SUBAPPLICATION Counter (* Subapplication Type *)
  (* Standard: 61499-2 *)
  (* Version 1.0, 2023-02-17, Franz *)
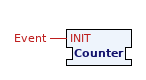
  EVENT_INPUT
    INIT;
  END_EVENT
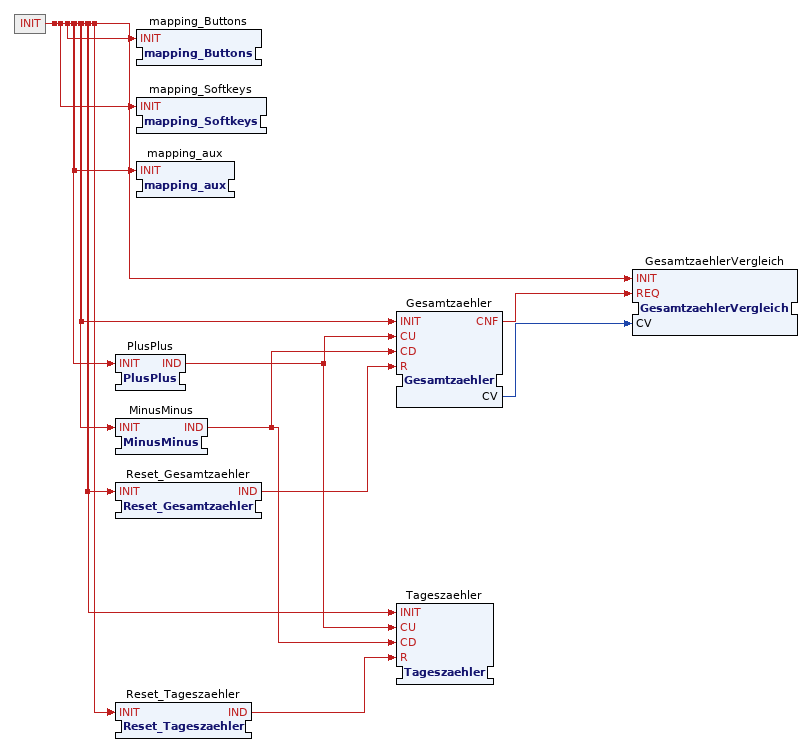
  SUBAPPS
    mapping_Buttons : mapping_Buttons;
    mapping_Softkeys : mapping_Softkeys;
    mapping_aux : mapping_aux;
    Gesamtzaehler : Gesamtzaehler;
    Tageszaehler : Tageszaehler;
    MinusMinus : MinusMinus;
    PlusPlus : PlusPlus;
    Reset_Gesamtzaehler : Reset_Gesamtzaehler;
    Reset_Tageszaehler : Reset_Tageszaehler;
    GesamtzaehlerVergleich : GesamtzaehlerVergleich;
  END_SUBAPPS
  EVENT_CONNECTIONS
    INIT TO mapping_Softkeys.INIT;
    INIT TO mapping_Buttons.INIT;
    INIT TO mapping_aux.INIT;
    INIT TO Gesamtzaehler.INIT;
    INIT TO Tageszaehler.INIT;
    PlusPlus.IND TO Gesamtzaehler.CU;
    PlusPlus.IND TO Tageszaehler.CU;
    MinusMinus.IND TO Gesamtzaehler.CD;
    MinusMinus.IND TO Tageszaehler.CD;
    INIT TO PlusPlus.INIT;
    INIT TO MinusMinus.INIT;
    INIT TO Reset_Gesamtzaehler.INIT;
    INIT TO Reset_Tageszaehler.INIT;
    Reset_Gesamtzaehler.IND TO Gesamtzaehler.R;
    Reset_Tageszaehler.IND TO Tageszaehler.R;
    INIT TO GesamtzaehlerVergleich.INIT;
    Gesamtzaehler.CNF TO GesamtzaehlerVergleich.REQ;
  END_CONNECTIONS
  DATA_CONNECTIONS
    Gesamtzaehler.CV TO GesamtzaehlerVergleich.CV;
  END_CONNECTIONS
END_SUBAPPLICATION
